(* CODESYS project Lypuny.project
   Title: Lypuny
   Author: d2581
   Version: 0.0.0.8

Project tree, tasks and I/O mapping:
  MyController : TM241CE40T/U, Schneider Electric, order no. TM241CE40T/U, version 4.0.6.18
    application Application
      task MAST (cyclic, interval 20 ms, priority 15, watchdog 100 ms x 1) calls nothing
      global variables GVL
      program Input [ST]
      program Output [ST]
    A1_IN : Digital Inputs, Schneider Electric, version 4.0.6.18
        input  idwDI_IDW0 : DWORD  // IDW0
        input  X0 : BOOL  // IDW0.I0
        input  X1 : BOOL  // IDW0.I1
        input  X2 : BOOL  // IDW0.I2
        input  X3 : BOOL  // IDW0.I3
        input  X4 : BOOL  // IDW0.I4
        input  X5 : BOOL  // IDW0.I5
        input  X6 : BOOL  // IDW0.I6
        input  X7 : BOOL  // IDW0.I7
        input  X8 : BOOL  // IDW0.I8
        input  X9 : BOOL  // IDW0.I9
        input  X10 : BOOL  // IDW0.I10
        input  X11 : BOOL  // IDW0.I11
        input  X12 : BOOL  // IDW0.I12
        input  X13 : BOOL  // IDW0.I13
        input  X14 : BOOL  // IDW0.I14
        input  X15 : BOOL  // IDW0.I15
        input  X16 : BOOL  // IDW0.I16
        input  X17 : BOOL  // IDW0.I17
        input  X18 : BOOL  // IDW0.I18
        input  X19 : BOOL  // IDW0.I19
        input  X20 : BOOL  // IDW0.I20
        input  X21 : BOOL  // IDW0.I21
        input  X22 : BOOL  // IDW0.I22
        input  X23 : BOOL  // IDW0.I23
        input  ibDI_IB1 : BYTE  // IB1
    A1_OUT : Digital Outputs, Schneider Electric, version 4.0.6.18
        output Y0 : BOOL  // QW0.Q0
        output Y1 : BOOL  // QW0.Q1
        output Y2 : BOOL  // QW0.Q2
        output Y3 : BOOL  // QW0.Q3
        output Y4 : BOOL  // QW0.Q4
        output Y5 : BOOL  // QW0.Q5
        output Y6 : BOOL  // QW0.Q6
        output Y7 : BOOL  // QW0.Q7
        output Y8 : BOOL  // QW0.Q8
        output Y9 : BOOL  // QW0.Q9
        output Y10 : BOOL  // QW0.Q10
        output Y11 : BOOL  // QW0.Q11
        output Y12 : BOOL  // QW0.Q12
        output Y13 : BOOL  // QW0.Q13
        output Y14 : BOOL  // QW0.Q14
        output Y15 : BOOL  // QW0.Q15
        output qbDQ_QB1 : BYTE  // QB1
        unmapped channels: QW0
    Counters : Counters, Schneider Electric, version 4.0.6.18
    Pulse_Generators : Pulse Generators, Schneider Electric, version 4.0.6.18
    Cartridge_1 : Cartridge, Schneider Electric, version 4.0.6.18
    Cartridge_2 : Cartridge, Schneider Electric, version 4.0.6.18
    IO_Bus : IO bus - TM3, Schneider Electric, version 4.0.6.18
      A1_1 : TM3DI16K, Schneider Electric, order no. TM3DI16K, version 1.0.1.4
          input  iwModule_1_IW0 : WORD  // IW0
          input  _1X0 : BOOL  // IW0.I0
          input  _1X1 : BOOL  // IW0.I1
          input  _1X2 : BOOL  // IW0.I2
          input  _1X3 : BOOL  // IW0.I3
          input  _1X4 : BOOL  // IW0.I4
          input  _1X5 : BOOL  // IW0.I5
          input  _1X6 : BOOL  // IW0.I6
          input  _1X7 : BOOL  // IW0.I7
          input  _1X8 : BOOL  // IW0.I8
          input  _1X9 : BOOL  // IW0.I9
          input  _1X10 : BOOL  // IW0.I10
          input  _1X11 : BOOL  // IW0.I11
          input  _1X12 : BOOL  // IW0.I12
          input  _1X13 : BOOL  // IW0.I13
          input  _1X14 : BOOL  // IW0.I14
          input  _1X15 : BOOL  // IW0.I15
      A1_2 : TM3DQ16TK, Schneider Electric, order no. TM3DQ16TK, version 1.0.1.4
          output _2Y0 : BOOL  // QW0.Q0
          output _2Y1 : BOOL  // QW0.Q1
          output _2Y2 : BOOL  // QW0.Q2
          output _2Y3 : BOOL  // QW0.Q3
          output _2Y4 : BOOL  // QW0.Q4
          output _2Y5 : BOOL  // QW0.Q5
          output _2Y6 : BOOL  // QW0.Q6
          output _2Y7 : BOOL  // QW0.Q7
          output _2Y8 : BOOL  // QW0.Q8
          output _2Y9 : BOOL  // QW0.Q9
          output _2Y10 : BOOL  // QW0.Q10
          output _2Y11 : BOOL  // QW0.Q11
          output _2Y12 : BOOL  // QW0.Q12
          output _2Y13 : BOOL  // QW0.Q13
          output _2Y14 : BOOL  // QW0.Q14
          output _2Y15 : BOOL  // QW0.Q15
          unmapped channels: QW0
      A1_3 : TM3AI4/G, Schneider Electric, order no. TM3AI4/G, version 1.0.0.15
          settings: KPI Configuration.KPI Configuration[0] = 35; KPI Configuration.KPI Configuration[1] = 35; KPI Configuration.KPI Configuration[2] = 35; KPI Configuration.KPI Configuration[3] = 35; KPI Configuration.KPI Configuration[4] = 160; KPI Configuration.KPI Configuration[5] = 15; KPI Configuration.KPI Configuration[6] = 160; KPI Configuration.KPI Configuration[7] = 15; KPI Configuration.KPI Configuration[8] = 160; KPI Configuration.KPI Configuration[9] = 15; KPI Configuration.KPI Configuration[10] = 160; KPI Configuration.KPI Configuration[11] = 15; KPI Configuration.KPI Configuration[12] = 32; KPI Configuration.KPI Configuration[13] = 78; KPI Configuration.KPI Configuration[14] = 32; KPI Configuration.KPI Configuration[15] = 78; KPI Configuration.KPI Configuration[16] = 32; KPI Configuration.KPI Configuration[17] = 78; KPI Configuration.KPI Configuration[18] = 32; KPI Configuration.KPI Configuration[19] = 78; KPI Configuration.KPI Configuration[20] = 1; KPI Configuration.KPI Configuration[22] = 1; KPI Configuration.KPI Configuration[24] = 1; KPI Configuration.KPI Configuration[26] = 1; KPI Configuration.KPI Configuration[29] = 1; KPI Configuration.KPI Configuration[30] = 1; KPI Configuration.KPI Configuration[31] = 1
          input  PE1 : INT  // IW0
          input  PE2 : INT  // IW1
          input  PE3 : INT  // IW2
          input  PERezerv : INT  // IW3
          input  ibModule_3_IBStatusIW0 : BYTE  // IBStatusIW0
          input  ibModule_3_IBStatusIW1 : BYTE  // IBStatusIW1
          input  ibModule_3_IBStatusIW2 : BYTE  // IBStatusIW2
          input  ibModule_3_IBStatusIW3 : BYTE  // IBStatusIW3
      A1_4 : TM3TI4/G, Schneider Electric, order no. TM3TI4/G, version 1.0.1.5
          settings: KPI Configuration.KPI Configuration[0] = 77; KPI Configuration.KPI Configuration[1] = 77; KPI Configuration.KPI Configuration[2] = 77; KPI Configuration.KPI Configuration[3] = 77; KPI Configuration.KPI Configuration[4] = 48; KPI Configuration.KPI Configuration[5] = 248; KPI Configuration.KPI Configuration[6] = 48; KPI Configuration.KPI Configuration[7] = 248; KPI Configuration.KPI Configuration[8] = 48; KPI Configuration.KPI Configuration[9] = 248; KPI Configuration.KPI Configuration[10] = 48; KPI Configuration.KPI Configuration[11] = 248; KPI Configuration.KPI Configuration[12] = 52; KPI Configuration.KPI Configuration[13] = 33; KPI Configuration.KPI Configuration[14] = 52; KPI Configuration.KPI Configuration[15] = 33; KPI Configuration.KPI Configuration[16] = 52; KPI Configuration.KPI Configuration[17] = 33; KPI Configuration.KPI Configuration[18] = 52; KPI Configuration.KPI Configuration[19] = 33; KPI Configuration.KPI Configuration[20] = 1; KPI Configuration.KPI Configuration[22] = 1; KPI Configuration.KPI Configuration[24] = 1; KPI Configuration.KPI Configuration[26] = 1
          input  TE1 : INT  // IW0
          input  TE2 : INT  // IW1
          input  TE3 : INT  // IW2
          input  TE4Rezerv : INT  // IW3
          input  ibModule_4_IBStatusIW0 : BYTE  // IBStatusIW0
          input  ibModule_4_IBStatusIW1 : BYTE  // IBStatusIW1
          input  ibModule_4_IBStatusIW2 : BYTE  // IBStatusIW2
          input  ibModule_4_IBStatusIW3 : BYTE  // IBStatusIW3
    COM_Bus : COM bus, Schneider Electric, version 4.0.6.18
    Ethernet_1 : Ethernet Network, Schneider Electric, version 4.0.6.18
    Serial_Line_1 : Serial line, Schneider Electric, version 4.0.6.18
      Modbus_Manager : Modbus Manager, Schneider Electric, version 4.0.0.2
    Serial_Line_2 : Serial line, Schneider Electric, version 4.0.6.18
*)

// MyController/Application/GVL
VAR_GLOBAL
	//------------------------------------------------------Inpup A1 A1.1 A1.3 A1.4-----------------------------------------
	Breake1 AT %MX0.0: BOOL;
	ErrBoiler1 AT %MX0.1: BOOL;
	ManualMode AT %MX0.2: BOOL;
	ErrBoiler2 AT %MX0.3: BOOL;
	Breake2 AT %MX0.4: BOOL;
	PressReversNetWtrLow AT %MX0.5: BOOL;
	PressReversNetWtrHigh AT %MX0.6: BOOL;
	DrySourceWtr1 AT %MX0.7: BOOL;
	PressSourceWtr1 AT %MX0.8: BOOL;
	DrySourceWtr2 AT %MX0.9: BOOL;
	PressSourceWtr2 AT %MX0.10: BOOL;
	DryNetWtr1 AT %MX0.11: BOOL;
	PressNetWtr1 AT %MX0.12: BOOL;
	DryNetWtr2 AT %MX0.13: BOOL;
	PressNetWtr2 AT %MX0.14: BOOL;
	DryFeederWtr1 AT %MX0.15: BOOL;
	PressFeederWtr1 AT %MX2.0: BOOL;
	DryFeederWtr2 AT %MX2.1: BOOL;//%MW1.1
	PressFeederWtr2 AT %MX2.2: BOOL;//%MW1.2
	PumpSourceWtr1On AT %MX2.3: BOOL;//%MW1.3
	PumpSourceWtr2On AT %MX2.4: BOOL;//%MW1.4
	PumpNetWtr1On AT %MX2.5: BOOL;//%MW1.5
	PumpNetWtr2On AT %MX2.6: BOOL;//%MW1.6
	PumpFeederWtr1On AT %MX2.7: BOOL;//%MW1.7
	PumpFeederWtr2On AT %MX2.8: BOOL;//%MW1.8
	ErrTopLevelReservTankWtr AT %MX2.9: BOOL;//%MW1.9
	TopLevelReservTankWtr AT %MX2.10: BOOL;//%MW1.10
	ErrLowLevelReservTankWtr AT %MX2.11: BOOL;//%MW1.11
	LowLevelReservTankWtr AT %MX2.12: BOOL;//%MW1.12
	Breake3 AT %MX2.13: BOOL;//%MW1.13
	// --------------------------------------------------------------резервные биты в слове -----------------------------------------------
	rezerv_mx2_13 AT %MX2.14: BOOL;
	rezerv_mx2_14 AT %MX2.15: BOOL;
	// -------------------------------------------------------------------------------------------------------------------------------------
	PressReversNetWtr AT %MD1: REAL;//%MW2,%MW3
	PE1Min AT %MW4: INT;
	PE1Max AT %MW5: INT;
	PressForwardNetWtr AT %MD3: REAL;//%MW6,%MW7
	PE2Min AT %MW8: INT;
	PE2Max AT %MW9: INT;
	PressSourceWtr AT %MD5: REAL;//%MW10,%MW11
	PE3Min AT %MW12: INT;
	PE3Max AT %MW13: INT;
	TpmReversNetWtr AT %MW14: INT;
	TmpAir AT %MW15: INT;
	TmpForwardWtr AT %MW16: INT;
	//------------------------------------------------------Outpun A1------------------------------------------------
	rezerv_mx34_0 AT %MX34.0: BOOL;
	PumpNetWtr1Run AT %MX34.1: BOOL;
	PumpNetWtr1Stop AT %MX34.2: BOOL;
	PumpNetWtr2Run AT %MX34.3: BOOL;
	PumpNetWtr2Stop AT %MX34.4: BOOL;
	PumpFeeder1Run AT %MX34.5: BOOL;
	PumpFeeder1Stop AT %MX34.6: BOOL;
	PumpFeeder2Run AT %MX34.7: BOOL;
	PumpFeeder2Stop AT %MX34.8: BOOL;
	PumpSourceWtr1Run AT %MX34.9: BOOL;
	PumpSourceWtr1Stop AT %MX34.10: BOOL;
	PumpSourceWtr2Run AT %MX34.11: BOOL;
	PumpSourceWtr2Stop AT %MX34.12: BOOL;
	VlvRezervTankWtrOpen AT %MX34.13: BOOL;
	RezervY13 AT %MX34.14: BOOL;
	VlvBypassOpen AT %MX34.15: BOOL;
	VlvBypassClose AT %MX36.0: BOOL;
	LightSignalColumn AT %MX36.1: BOOL;
	// --------------------------------------------------3 реле в резерве-----------------------------------------------
	Rezerv2Y1 AT %MX36.2: BOOL;
	Rezerv2Y2 AT %MX36.3: BOOL;
	Rezerv2Y3 AT %MX36.4: BOOL;
	// --------------------------------------------------резервные биты в слове-----------------------------------------
	rezerv_mx36_5 AT %MX36.5: BOOL;
	rezerv_mx36_6 AT %MX36.6: BOOL;
	rezerv_mx36_7 AT %MX36.7: BOOL;
	rezerv_mx36_8 AT %MX36.8: BOOL;
	rezerv_mx36_9 AT %MX36.9: BOOL;
	rezerv_mx36_10 AT %MX36.10: BOOL;
	rezerv_mx36_11 AT %MX36.11: BOOL;
	rezerv_mx36_12 AT %MX36.12: BOOL;
	rezerv_mx36_13 AT %MX36.13: BOOL;
	rezerv_mx36_14 AT %MX36.14: BOOL;
	rezerv_mx36_15 AT %MX36.15: BOOL;
	// -----------------------------------------------------------------------------------------------------------------
END_VAR

// MyController/Application/Input
PROGRAM Input
VAR

END_VAR

Breake1 := NOT X0;
ErrBoiler1 := X1;
ManualMode := X2;
ErrBoiler2 := X3;
Breake2 := NOT X4;
PressReversNetWtrLow := NOT X5;//PIS9
PressReversNetWtrHigh := X6;//PIS9
DrySourceWtr1 := NOT X7;//PIS7
PressSourceWtr1 := X8;//PIS5
DrySourceWtr2 := NOT X9;//PIS8
PressSourceWtr2 := NOT X10;//PIS6
DryNetWtr1 := NOT X11;//PIS3
PressNetWtr1 := NOT X12;//PIS1
DryNetWtr2 := NOT X13;//PIS4
PressNetWtr2 := NOT X14;//PIS2
DryFeederWtr1 := NOT X15;//PIS11
PressFeederWtr1 := NOT X16; //PIS9
DryFeederWtr2 := NOT X17;//PIS12
PressFeederWtr2 := NOT X18; //PIS12
PumpSourceWtr1On := X19;//KM-K6.1
PumpSourceWtr2On := X20;//KM-K6.2
PumpNetWtr1On := X21;//KM-K3.1
PumpNetWtr2On := X22;//KM-K3.2
PumpFeederWtr1On := X23;//KM-K4.1
PumpFeederWtr2On := _1X0;//KM-K4.2
ErrTopLevelReservTankWtr := _1X1;//Верхний аварийный уровень в баке запаса воды
TopLevelReservTankWtr := _1X2;//Верхний рабочий уровень в баке запаса воды
ErrLowLevelReservTankWtr := _1X3;//Нижний аварийный уровень в баке запаса воды
LowLevelReservTankWtr := _1X4;//Нижний рабочий уровень в баке запаса воды
Breake3 := NOT _1X5;
PressReversNetWtr := LIN_TRAFO(PE1, 4000, 20000, PE1Min, PE1Max);//Давление обратной сетевой воды
PressForwardNetWtr := LIN_TRAFO(PE2, 4000, 20000, PE2Min, PE2Max);//Давление прямой сетевой воды 
PressSourceWtr := LIN_TRAFO(PE3, 4000, 20000, PE3Min, PE3Max);//Давление прямой сетевой воды 
TpmReversNetWtr := TE1;//Температура обратной сетевой воды на входе в котельную
TmpForwardWtr := TE2;//Температура прямой сетевой воды на выходе из котельной
TmpAir := TE3;//Температура наружнего воздуха

END_PROGRAM

// MyController/Application/Output
PROGRAM Output
VAR	
END_VAR

Y0 := PumpNetWtr1Run;
Y1 := NOT PumpNetWtr1Stop;
Y2 := PumpNetWtr2Run;
Y3 := NOT PumpNetWtr2Stop;
Y4 := PumpFeeder1Run;
Y5 := NOT PumpFeeder1Stop;
Y6 :=  PumpFeeder2Run;
Y7 := NOT PumpFeeder2Stop;
Y8 := PumpSourceWtr1Run;
Y9 := NOT PumpSourceWtr1Stop;
Y10 := PumpSourceWtr2Run;
Y11 := NOT PumpSourceWtr2Stop;
Y12 := VlvRezervTankWtrOpen;
Y13 := RezervY13;
Y14 := VlvBypassOpen;
Y15 := VlvBypassClose;
_2Y0 := LightSignalColumn;
_2Y1 := Rezerv2Y1;
_2Y2 := Rezerv2Y2;
_2Y3 := Rezerv2Y3;

END_PROGRAM
